// TIA Portal V20 export
TYPE "LConSMC_typeWebbreakDetectDiag"
// Diagnose der Bahnrisserkennung / Diagnostic structre for webbreak detection
// stored: Access Published
   STRUCT
      webbreakDetectionActive : Bool;   // TRUE: Die Bahnrissüberwachung ist aktiv / TRUE: Web break detection is active
      webBreak : Bool;   // TRUE: Es wurde ein Bahnriss erkannt Der PID-Regler wird deaktiviert / TRUE: A web break has been detected. The PID controlled will be disabled
   END_STRUCT;
END_TYPE
